(* IEC 61131-3 sources: eCockpitGit/test_project/src/%F%02 System/%F%03 LoadSaveManager/%POU%FB_LoadSave/%F%Load/%F%Structure/%PRO%selectedType, 1 file *)

(* ---- %GETSET%Get.st ---- *)
VAR
END_VAR

(*%!%__DELIMITER__%!%*)
selectedType	:=		reader.selectedType;
